// TIA Portal V19 export
TYPE "C501_VAR_IF_TME_TYPIC"
   STRUCT
      MWA { ExternalAccessible := 'False'; ExternalVisible := 'False'; ExternalWritable := 'False'} : Real;   // Meetwaarde
      EXT_HW { ExternalAccessible := 'False'; ExternalVisible := 'False'; ExternalWritable := 'False'} : Bool;   // Sturings hardware (PLC) in storing
      STO { ExternalAccessible := 'False'; ExternalVisible := 'False'; ExternalWritable := 'False'} : Struct   // Opsomming van alle storingen
         A001 : Bool;   // Beveiliging aangesproken
         A002 : Bool;   // Draadbreuk analoge meting
         A003 : Bool;   // Meetbereik overschreden
         A004 : Bool;   // Temperatuurmeter geeft storing
      END_STRUCT;
   END_STRUCT;
END_TYPE
